  [299] = "0.269000,-22.048000,213.211000,-177.000000,0.007000,-179.714000,"
  [300] = "-1.345000,-22.065000,213.211000,-177.000000,-0.037000,178.570000,"
  [301] = "-2.959000,-22.137000,213.210000,-177.000000,-0.082000,176.853000,"
  [302] = "-4.573000,-22.261000,213.210000,-177.000000,-0.128000,175.133000,"
  [303] = "-6.186000,-22.440000,213.210000,-177.000000,-0.173000,173.409000,"
  [304] = "-7.799000,-22.673000,213.209000,-177.000000,-0.218000,171.678000,"
  [305] = "-9.410000,-22.962000,213.208000,-177.000000,-0.264000,169.940000,"
  [306] = "-11.020000,-23.306000,213.207000,-177.000000,-0.310000,168.192000,"
  [307] = "-12.628000,-23.707000,213.206000,-177.000000,-0.357000,166.434000,"
  [308] = "-14.234000,-24.166000,213.205000,-177.000000,-0.404000,164.662000,"
  [309] = "-15.838000,-24.685000,213.204000,-177.000000,-0.452000,162.874000,"
  [310] = "-17.439000,-25.265000,213.203000,-177.000000,-0.500000,161.070000,"
  [311] = "-17.459000,-25.264000,210.801000,-177.000000,-0.500000,161.072000,"
  [312] = "-17.480000,-25.264000,208.203000,-177.000000,-0.500000,161.074000,"
  [313] = "-16.142000,-24.776000,208.204000,-177.000000,-0.460000,162.579000,"
  [314] = "-14.535000,-24.248000,208.205000,-177.000000,-0.412000,164.368000,"
  [315] = "-12.925000,-23.779000,208.206000,-177.000000,-0.365000,166.142000,"
  [316] = "-11.313000,-23.368000,208.207000,-177.000000,-0.318000,167.903000,"
  [317] = "-9.700000,-23.015000,208.208000,-177.000000,-0.272000,169.652000,"
  [318] = "-8.085000,-22.717000,208.209000,-177.000000,-0.226000,171.391000,"
  [319] = "-6.470000,-22.475000,208.210000,-177.000000,-0.180000,173.122000,"
  [320] = "-4.853000,-22.287000,208.210000,-177.000000,-0.135000,174.847000,"
  [321] = "-3.236000,-22.154000,208.210000,-177.000000,-0.090000,176.567000,"
  [322] = "-1.618000,-22.074000,208.211000,-177.000000,-0.045000,178.284000,"
  [323] = "0.000000,-22.047000,208.211000,-177.000000,0.000000,180.000000,"
  [324] = "1.618000,-22.074000,208.211000,-177.000000,0.045000,-178.284000,"
  [325] = "3.236000,-22.154000,208.210000,-177.000000,0.090000,-176.567000,"
  [326] = "4.853000,-22.287000,208.210000,-177.000000,0.135000,-174.847000,"
  [327] = "6.470000,-22.475000,208.210000,-177.000000,0.180000,-173.122000,"
  [328] = "8.085000,-22.717000,208.209000,-177.000000,0.226000,-171.391000,"
  [329] = "9.700000,-23.015000,208.208000,-177.000000,0.272000,-169.651000,"
  [330] = "11.313000,-23.368000,208.207000,-177.000000,0.318000,-167.902000,"
  [331] = "12.925000,-23.779000,208.206000,-177.000000,0.365000,-166.142000,"
  [332] = "14.535000,-24.248000,208.205000,-177.000000,0.412000,-164.368000,"
  [333] = "16.142000,-24.776000,208.204000,-177.000000,0.460000,-162.579000,"
  [334] = "17.480000,-25.264000,208.203000,-177.000000,0.500000,-161.074000,"
  [335] = "17.502000,-25.264000,205.801000,-177.000000,0.500000,-161.072000,"
  [336] = "17.527000,-25.265000,203.203000,-177.000000,0.500000,-161.070000,"
  [337] = "15.929000,-24.689000,203.204000,-177.000000,0.452000,-162.861000,"
  [338] = "14.329000,-24.174000,203.206000,-177.000000,0.405000,-164.635000,"
  [339] = "12.727000,-23.717000,203.207000,-177.000000,0.358000,-166.393000,"
  [340] = "11.123000,-23.317000,203.208000,-177.000000,0.312000,-168.139000,"
  [341] = "9.518000,-22.974000,203.208000,-177.000000,0.266000,-169.874000,"
  [342] = "7.911000,-22.685000,203.209000,-177.000000,0.220000,-171.599000,"
  [343] = "6.303000,-22.451000,203.210000,-177.000000,0.175000,-173.316000,"
  [344] = "4.695000,-22.271000,203.210000,-177.000000,0.130000,-175.028000,"
  [345] = "3.085000,-22.144000,203.210000,-177.000000,0.086000,-176.735000,"
  [346] = "1.476000,-22.069000,203.211000,-177.000000,0.041000,-178.439000,"
  [347] = "0.134000,-22.047000,203.211000,-177.000000,0.004000,-179.858000,"
  [348] = "-1.476000,-22.069000,203.211000,-177.000000,-0.041000,178.439000,"
  [349] = "-3.085000,-22.144000,203.210000,-177.000000,-0.086000,176.735000,"
  [350] = "-4.695000,-22.271000,203.210000,-177.000000,-0.130000,175.028000,"
  [351] = "-6.303000,-22.451000,203.210000,-177.000000,-0.175000,173.316000,"
  [352] = "-7.911000,-22.685000,203.209000,-177.000000,-0.220000,171.599000,"
  [353] = "-9.518000,-22.974000,203.208000,-177.000000,-0.266000,169.874000,"
  [354] = "-11.123000,-23.317000,203.208000,-177.000000,-0.312000,168.139000,"
  [355] = "-12.727000,-23.717000,203.207000,-177.000000,-0.358000,166.393000,"
  [356] = "-14.329000,-24.174000,203.206000,-177.000000,-0.405000,164.635000,"
  [357] = "-15.929000,-24.689000,203.204000,-177.000000,-0.452000,162.861000,"
  [358] = "-17.527000,-25.265000,203.203000,-177.000000,-0.500000,161.070000,"
  [359] = "-17.546000,-25.264000,200.801000,-177.000000,-0.500000,161.072000,"
  [360] = "-17.567000,-25.264000,198.203000,-177.000000,-0.500000,161.074000,"
  [361] = "-15.966000,-24.688000,198.204000,-177.000000,-0.452000,162.864000,"
  [362] = "-14.362000,-24.173000,198.206000,-177.000000,-0.405000,164.638000,"
  [363] = "-12.756000,-23.716000,198.207000,-177.000000,-0.358000,166.396000,"
  [364] = "-11.148000,-23.317000,198.208000,-177.000000,-0.312000,168.141000,"
  [365] = "-9.539000,-22.973000,198.208000,-177.000000,-0.266000,169.876000,"
  [366] = "-7.929000,-22.685000,198.209000,-177.000000,-0.220000,171.600000,"
  [367] = "-6.317000,-22.451000,198.210000,-177.000000,-0.175000,173.318000,"
  [368] = "-4.705000,-22.271000,198.210000,-177.000000,-0.130000,175.029000,"
  [369] = "-3.092000,-22.143000,198.210000,-177.000000,-0.086000,176.736000,"
  [370] = "-1.479000,-22.069000,198.211000,-177.000000,-0.041000,178.439000,"
  [371] = "-0.134000,-22.047000,198.211000,-177.000000,-0.004000,179.858000,"
  [372] = "1.479000,-22.069000,198.211000,-177.000000,0.041000,-178.439000,"
  [373] = "3.092000,-22.143000,198.210000,-177.000000,0.086000,-176.736000,"
  [374] = "4.705000,-22.271000,198.210000,-177.000000,0.130000,-175.029000,"
  [375] = "6.317000,-22.451000,198.210000,-177.000000,0.175000,-173.318000,"
  [376] = "7.929000,-22.685000,198.209000,-177.000000,0.220000,-171.600000,"
  [377] = "9.539000,-22.973000,198.208000,-177.000000,0.266000,-169.875000,"
  [378] = "11.148000,-23.317000,198.208000,-177.000000,0.312000,-168.141000,"
  [379] = "12.756000,-23.716000,198.207000,-177.000000,0.358000,-166.396000,"
  [380] = "14.362000,-24.173000,198.206000,-177.000000,0.405000,-164.638000,"
  [381] = "15.966000,-24.688000,198.204000,-177.000000,0.452000,-162.864000,"
  [382] = "17.567000,-25.264000,198.203000,-177.000000,0.500000,-161.074000,"
  [383] = "17.590000,-25.264000,195.801000,-177.000000,0.500000,-161.072000,"
  [384] = "17.614000,-25.265000,193.203000,-177.000000,0.500000,-161.070000,"
  [385] = "16.008000,-24.689000,193.205000,-177.000000,0.452000,-162.861000,"
  [386] = "14.400000,-24.174000,193.206000,-177.000000,0.405000,-164.635000,"
  [387] = "12.790000,-23.717000,193.207000,-177.000000,0.358000,-166.393000,"
  [388] = "11.178000,-23.317000,193.208000,-177.000000,0.312000,-168.139000,"
  [389] = "9.564000,-22.974000,193.209000,-177.000000,0.266000,-169.874000,"
  [390] = "7.949000,-22.685000,193.209000,-177.000000,0.220000,-171.599000,"
  [391] = "6.334000,-22.451000,193.210000,-177.000000,0.175000,-173.316000,"
  [392] = "4.717000,-22.271000,193.210000,-177.000000,0.130000,-175.028000,"
  [393] = "3.100000,-22.143000,193.210000,-177.000000,0.086000,-176.735000,"
  [394] = "1.483000,-22.069000,193.211000,-177.000000,0.041000,-178.439000,"
  [395] = "0.135000,-22.047000,193.211000,-177.000000,0.004000,-179.858000,"
  [396] = "-1.483000,-22.069000,193.211000,-177.000000,-0.041000,178.439000,"
  [397] = "-3.100000,-22.144000,193.210000,-177.000000,-0.086000,176.735000,"
  [398] = "-4.717000,-22.271000,193.210000,-177.000000,-0.130000,175.028000,"
  [399] = "-6.334000,-22.451000,193.210000,-177.000000,-0.175000,173.316000,"
  [400] = "-7.949000,-22.685000,193.209000,-177.000000,-0.220000,171.599000,"
  [401] = "-9.564000,-22.974000,193.209000,-177.000000,-0.266000,169.874000,"
  [402] = "-11.178000,-23.317000,193.208000,-177.000000,-0.312000,168.139000,"
  [403] = "-12.790000,-23.717000,193.207000,-177.000000,-0.358000,166.393000,"
  [404] = "-14.400000,-24.174000,193.206000,-177.000000,-0.405000,164.635000,"
  [405] = "-16.008000,-24.689000,193.205000,-177.000000,-0.452000,162.861000,"
  [406] = "-17.614000,-25.265000,193.203000,-177.000000,-0.500000,161.070000,"
  [407] = "-17.633000,-25.264000,190.801000,-177.000000,-0.500000,161.072000,"
  [408] = "-17.654000,-25.264000,188.204000,-177.000000,-0.500000,161.074000,"
  [409] = "-16.057000,-24.692000,188.205000,-177.000000,-0.452000,162.851000,"
  [410] = "-14.457000,-24.180000,188.206000,-177.000000,-0.405000,164.611000,"
  [411] = "-12.855000,-23.726000,188.207000,-177.000000,-0.359000,166.356000,"
  [412] = "-11.252000,-23.328000,188.208000,-177.000000,-0.313000,168.089000,"
  [413] = "-9.647000,-22.985000,188.209000,-177.000000,-0.268000,169.810000,"
  [414] = "-8.041000,-22.697000,188.209000,-177.000000,-0.222000,171.522000,"
  [415] = "-6.434000,-22.462000,188.210000,-177.000000,-0.178000,173.227000,"
  [416] = "-4.826000,-22.280000,188.210000,-177.000000,-0.133000,174.925000,"
  [417] = "-3.218000,-22.150000,188.210000,-177.000000,-0.089000,176.619000,"
  [418] = "-1.609000,-22.073000,188.211000,-177.000000,-0.044000,178.310000,"
  [419] = "0.000000,-22.047000,188.211000,-177.000000,0.000000,180.000000,"
  [420] = "1.609000,-22.073000,188.211000,-177.000000,0.044000,-178.310000,"
  [421] = "3.218000,-22.150000,188.210000,-177.000000,0.089000,-176.619000,"
  [422] = "4.826000,-22.280000,188.210000,-177.000000,0.133000,-174.925000,"
  [423] = "6.434000,-22.462000,188.210000,-177.000000,0.178000,-173.227000,"
  [424] = "8.041000,-22.697000,188.209000,-177.000000,0.222000,-171.522000,"
  [425] = "9.647000,-22.985000,188.209000,-177.000000,0.268000,-169.810000,"
  [426] = "11.252000,-23.328000,188.208000,-177.000000,0.313000,-168.089000,"
  [427] = "12.855000,-23.726000,188.207000,-177.000000,0.359000,-166.356000,"
  [428] = "14.457000,-24.180000,188.206000,-177.000000,0.405000,-164.611000,"
  [429] = "16.057000,-24.692000,188.205000,-177.000000,0.452000,-162.851000,"
  [430] = "17.654000,-25.264000,188.204000,-177.000000,0.500000,-161.074000,"
  [431] = "17.677000,-25.264000,185.801000,-177.000000,0.500000,-161.072000,"
  [432] = "17.702000,-25.265000,183.204000,-177.000000,0.500000,-161.070000,"
  [433] = "16.099000,-24.693000,183.205000,-177.000000,0.453000,-162.847000,"
  [434] = "14.495000,-24.181000,183.206000,-177.000000,0.406000,-164.608000,"
  [435] = "12.889000,-23.727000,183.207000,-177.000000,0.359000,-166.354000,"
  [436] = "11.281000,-23.329000,183.208000,-177.000000,0.313000,-168.086000,"
  [437] = "9.672000,-22.986000,183.209000,-177.000000,0.268000,-169.808000,"
  [438] = "8.062000,-22.697000,183.209000,-177.000000,0.222000,-171.521000,"
  [439] = "6.450000,-22.462000,183.210000,-177.000000,0.178000,-173.225000,"
  [440] = "4.839000,-22.280000,183.210000,-177.000000,0.133000,-174.924000,"
  [441] = "3.226000,-22.151000,183.210000,-177.000000,0.089000,-176.619000,"
  [442] = "1.613000,-22.073000,183.211000,-177.000000,0.044000,-178.310000,"
  [443] = "0.000000,-22.047000,183.211000,-177.000000,0.000000,180.000000,"
  [444] = "-1.613000,-22.073000,183.211000,-177.000000,-0.044000,178.310000,"
  [445] = "-3.226000,-22.151000,183.210000,-177.000000,-0.089000,176.619000,"
  [446] = "-4.838000,-22.280000,183.210000,-177.000000,-0.133000,174.924000,"
  [447] = "-6.450000,-22.462000,183.210000,-177.000000,-0.178000,173.225000,"
  [448] = "-8.062000,-22.697000,183.209000,-177.000000,-0.222000,171.521000,"
  [449] = "-9.672000,-22.986000,183.209000,-177.000000,-0.268000,169.808000,"
  [450] = "-11.281000,-23.329000,183.208000,-177.000000,-0.313000,168.086000,"
  [451] = "-12.889000,-23.727000,183.207000,-177.000000,-0.359000,166.354000,"
  [452] = "-14.495000,-24.181000,183.206000,-177.000000,-0.406000,164.608000,"
  [453] = "-16.099000,-24.693000,183.205000,-177.000000,-0.453000,162.847000,"
  [454] = "-17.701000,-25.265000,183.204000,-177.000000,-0.500000,161.070000,"
  [455] = "-17.721000,-25.264000,180.802000,-177.000000,-0.500000,161.072000,"
  [456] = "-17.742000,-25.264000,178.204000,-177.000000,-0.500000,161.074000,"
  [457] = "-16.136000,-24.692000,178.205000,-177.000000,-0.452000,162.851000,"
  [458] = "-14.528000,-24.180000,178.206000,-177.000000,-0.405000,164.611000,"
  [459] = "-12.918000,-23.726000,178.207000,-177.000000,-0.359000,166.356000,"
  [460] = "-11.306000,-23.328000,178.208000,-177.000000,-0.313000,168.089000,"
  [461] = "-9.693000,-22.985000,178.209000,-177.000000,-0.268000,169.810000,"
  [462] = "-8.080000,-22.697000,178.209000,-177.000000,-0.222000,171.522000,"
  [463] = "-6.465000,-22.462000,178.210000,-177.000000,-0.178000,173.227000,"
  [464] = "-4.849000,-22.280000,178.210000,-177.000000,-0.133000,174.925000,"
  [465] = "-3.233000,-22.150000,178.210000,-177.000000,-0.089000,176.619000,"
  [466] = "-1.617000,-22.073000,178.211000,-177.000000,-0.044000,178.310000,"
  [467] = "0.000000,-22.047000,178.211000,-177.000000,0.000000,180.000000,"
  [468] = "1.617000,-22.073000,178.211000,-177.000000,0.044000,-178.310000,"
  [469] = "3.233000,-22.150000,178.210000,-177.000000,0.089000,-176.619000,"
  [470] = "4.849000,-22.280000,178.210000,-177.000000,0.133000,-174.925000,"
  [471] = "6.465000,-22.462000,178.210000,-177.000000,0.178000,-173.227000,"
  [472] = "8.080000,-22.697000,178.209000,-177.000000,0.222000,-171.522000,"
  [473] = "9.694000,-22.985000,178.209000,-177.000000,0.268000,-169.810000,"
  [474] = "11.306000,-23.328000,178.208000,-177.000000,0.313000,-168.089000,"
  [475] = "12.918000,-23.726000,178.207000,-177.000000,0.359000,-166.356000,"
  [476] = "14.528000,-24.180000,178.206000,-177.000000,0.405000,-164.611000,"
  [477] = "16.136000,-24.692000,178.205000,-177.000000,0.452000,-162.851000,"
  [478] = "17.742000,-25.264000,178.204000,-177.000000,0.500000,-161.074000,"
  [479] = "17.764000,-25.264000,175.802000,-177.000000,0.500000,-161.072000,"
  [480] = "17.789000,-25.265000,173.204000,-177.000000,0.500000,-161.070000,"
  [481] = "16.178000,-24.693000,173.205000,-177.000000,0.453000,-162.848000,"
  [482] = "14.566000,-24.181000,173.206000,-177.000000,0.406000,-164.608000,"
  [483] = "12.952000,-23.727000,173.207000,-177.000000,0.359000,-166.354000,"
  [484] = "11.336000,-23.329000,173.208000,-177.000000,0.313000,-168.086000,"
  [485] = "9.719000,-22.986000,173.209000,-177.000000,0.268000,-169.808000,"
  [486] = "8.101000,-22.697000,173.209000,-177.000000,0.222000,-171.521000,"
  [487] = "6.481000,-22.462000,173.210000,-177.000000,0.178000,-173.225000,"
  [488] = "4.862000,-22.280000,173.210000,-177.000000,0.133000,-174.924000,"
  [489] = "3.241000,-22.150000,173.210000,-177.000000,0.089000,-176.619000,"
  [490] = "1.621000,-22.073000,173.211000,-177.000000,0.044000,-178.310000,"
  [491] = "0.000000,-22.047000,173.211000,-177.000000,0.000000,180.000000,"
  [492] = "-1.621000,-22.073000,173.211000,-177.000000,-0.044000,178.310000,"
  [493] = "-3.241000,-22.151000,173.210000,-177.000000,-0.089000,176.619000,"
  [494] = "-4.862000,-22.280000,173.210000,-177.000000,-0.133000,174.924000,"
  [495] = "-6.481000,-22.462000,173.210000,-177.000000,-0.178000,173.225000,"
  [496] = "-8.101000,-22.697000,173.209000,-177.000000,-0.222000,171.521000,"
  [497] = "-9.719000,-22.986000,173.209000,-177.000000,-0.268000,169.808000,"
  [498] = "-11.336000,-23.329000,173.208000,-177.000000,-0.313000,168.086000,"
  [499] = "-12.952000,-23.727000,173.207000,-177.000000,-0.359000,166.354000,"
  [500] = "-14.566000,-24.181000,173.206000,-177.000000,-0.406000,164.608000,"
  [501] = "-16.178000,-24.693000,173.205000,-177.000000,-0.453000,162.848000,"
  [502] = "-17.789000,-25.265000,173.204000,-177.000000,-0.500000,161.070000,"
  [503] = "-17.808000,-25.264000,170.802000,-177.000000,-0.500000,161.072000,"
  [504] = "-17.829000,-25.264000,168.204000,-177.000000,-0.500000,161.074000,"
  [505] = "-16.227000,-24.696000,168.205000,-177.000000,-0.453000,162.838000,"
  [506] = "-14.623000,-24.188000,168.206000,-177.000000,-0.406000,164.585000,"
  [507] = "-13.017000,-23.736000,168.207000,-177.000000,-0.360000,166.317000,"
  [508] = "-11.410000,-23.339000,168.208000,-177.000000,-0.314000,168.037000,"
  [509] = "-9.801000,-22.997000,168.209000,-177.000000,-0.269000,169.746000,"
  [510] = "-8.192000,-22.709000,168.209000,-177.000000,-0.224000,171.445000,"
  [511] = "-6.581000,-22.473000,168.210000,-177.000000,-0.180000,173.137000,"
  [512] = "-4.970000,-22.290000,168.210000,-177.000000,-0.136000,174.823000,"
  [513] = "-3.358000,-22.158000,168.210000,-177.000000,-0.092000,176.505000,"
  [514] = "-1.746000,-22.077000,168.211000,-177.000000,-0.048000,178.183000,"
  [515] = "-0.672000,-22.051000,168.211000,-177.000000,-0.018000,179.301000,"
  [516] = "0.134000,-22.047000,168.211000,-177.000000,0.004000,-179.860000,"
  [517] = "1.747000,-22.077000,168.211000,-177.000000,0.048000,-178.183000,"
  [518] = "3.358000,-22.158000,168.210000,-177.000000,0.092000,-176.505000,"
  [519] = "4.970000,-22.290000,168.210000,-177.000000,0.136000,-174.823000,"
  [520] = "6.581000,-22.473000,168.210000,-177.000000,0.180000,-173.137000,"
  [521] = "8.192000,-22.709000,168.209000,-177.000000,0.224000,-171.445000,"
  [522] = "9.801000,-22.997000,168.209000,-177.000000,0.269000,-169.746000,"
  [523] = "11.410000,-23.339000,168.208000,-177.000000,0.314000,-168.037000,"
  [524] = "13.017000,-23.736000,168.207000,-177.000000,0.360000,-166.317000,"
  [525] = "14.623000,-24.188000,168.206000,-177.000000,0.406000,-164.585000,"
  [526] = "16.227000,-24.696000,168.205000,-177.000000,0.453000,-162.838000,"
  [527] = "17.829000,-25.264000,168.204000,-177.000000,0.500000,-161.074000,"
  [528] = "17.852000,-25.264000,165.802000,-177.000000,0.500000,-161.072000,"
  [529] = "17.876000,-25.265000,163.204000,-177.000000,0.500000,-161.070000,"
  [530] = "16.270000,-24.697000,163.206000,-177.000000,0.453000,-162.834000,"
  [531] = "14.661000,-24.188000,163.207000,-177.000000,0.406000,-164.582000,"
  [532] = "13.051000,-23.736000,163.207000,-177.000000,0.360000,-166.314000,"
  [533] = "11.439000,-23.340000,163.208000,-177.000000,0.314000,-168.034000,"
  [534] = "9.827000,-22.998000,163.209000,-177.000000,0.269000,-169.744000,"
  [535] = "8.213000,-22.709000,163.209000,-177.000000,0.224000,-171.444000,"
  [536] = "6.598000,-22.473000,163.210000,-177.000000,0.180000,-173.136000,"
  [537] = "4.983000,-22.290000,163.210000,-177.000000,0.136000,-174.822000,"
  [538] = "3.367000,-22.158000,163.210000,-177.000000,0.092000,-176.504000,"
  [539] = "1.751000,-22.077000,163.211000,-177.000000,0.048000,-178.183000,"
  [540] = "0.673000,-22.051000,163.211000,-177.000000,0.018000,-179.301000,"
  [541] = "-0.135000,-22.047000,163.211000,-177.000000,-0.004000,179.860000,"
  [542] = "-1.751000,-22.077000,163.211000,-177.000000,-0.048000,178.183000,"
  [543] = "-3.367000,-22.158000,163.210000,-177.000000,-0.092000,176.504000,"
  [544] = "-4.983000,-22.290000,163.210000,-177.000000,-0.136000,174.822000,"
  [545] = "-6.598000,-22.473000,163.210000,-177.000000,-0.180000,173.136000,"
  [546] = "-8.213000,-22.709000,163.209000,-177.000000,-0.224000,171.444000,"
  [547] = "-9.827000,-22.998000,163.209000,-177.000000,-0.269000,169.744000,"
  [548] = "-11.439000,-23.340000,163.208000,-177.000000,-0.314000,168.034000,"
  [549] = "-13.051000,-23.736000,163.207000,-177.000000,-0.360000,166.314000,"
  [550] = "-14.661000,-24.188000,163.207000,-177.000000,-0.406000,164.582000,"
  [551] = "-16.270000,-24.697000,163.206000,-177.000000,-0.453000,162.834000,"
  [552] = "-17.876000,-25.265000,163.204000,-177.000000,-0.500000,161.070000,"
  [553] = "-17.896000,-25.264000,160.802000,-177.000000,-0.500000,161.072000,"
  [554] = "-17.917000,-25.264000,158.205000,-177.000000,-0.500000,161.074000,"
  [555] = "-16.306000,-24.696000,158.206000,-177.000000,-0.453000,162.838000,"
  [556] = "-14.694000,-24.188000,158.207000,-177.000000,-0.406000,164.585000,"
  [557] = "-13.080000,-23.736000,158.208000,-177.000000,-0.360000,166.317000,"
  [558] = "-11.465000,-23.339000,158.208000,-177.000000,-0.314000,168.037000,"
  [559] = "-9.848000,-22.997000,158.209000,-177.000000,-0.269000,169.746000,"
  [560] = "-8.231000,-22.709000,158.209000,-177.000000,-0.224000,171.445000,"
  [561] = "-6.613000,-22.473000,158.210000,-177.000000,-0.180000,173.137000,"
  [562] = "-4.994000,-22.290000,158.210000,-177.000000,-0.136000,174.823000,"
  [563] = "-3.374000,-22.158000,158.210000,-177.000000,-0.092000,176.505000,"
  [564] = "-1.755000,-22.077000,158.211000,-177.000000,-0.048000,178.183000,"
  [565] = "-0.675000,-22.051000,158.211000,-177.000000,-0.018000,179.301000,"
  [566] = "0.135000,-22.047000,158.211000,-177.000000,0.004000,-179.860000,"
  [567] = "1.755000,-22.077000,158.211000,-177.000000,0.048000,-178.183000,"
  [568] = "3.374000,-22.158000,158.210000,-177.000000,0.092000,-176.505000,"
  [569] = "4.994000,-22.290000,158.210000,-177.000000,0.136000,-174.823000,"
  [570] = "6.613000,-22.473000,158.210000,-177.000000,0.180000,-173.137000,"
  [571] = "8.231000,-22.709000,158.209000,-177.000000,0.224000,-171.445000,"
  [572] = "9.848000,-22.997000,158.209000,-177.000000,0.269000,-169.746000,"
  [573] = "11.465000,-23.339000,158.208000,-177.000000,0.314000,-168.037000,"
  [574] = "13.080000,-23.736000,158.208000,-177.000000,0.360000,-166.317000,"
  [575] = "14.694000,-24.188000,158.207000,-177.000000,0.406000,-164.585000,"
  [576] = "16.306000,-24.696000,158.206000,-177.000000,0.453000,-162.838000,"
  [577] = "17.917000,-25.264000,158.205000,-177.000000,0.500000,-161.074000,"
  [578] = "17.939000,-25.264000,155.803000,-177.000000,0.500000,-161.072000,"
  [579] = "17.964000,-25.265000,153.205000,-177.000000,0.500000,-161.070000,"
  [580] = "16.361000,-24.701000,153.206000,-177.000000,0.453000,-162.821000,"
  [581] = "14.756000,-24.196000,153.207000,-177.000000,0.407000,-164.556000,"
  [582] = "13.150000,-23.746000,153.208000,-177.000000,0.361000,-166.276000,"
  [583] = "11.543000,-23.351000,153.208000,-177.000000,0.316000,-167.983000,"
  [584] = "9.934000,-23.010000,153.209000,-177.000000,0.271000,-169.680000,"
  [585] = "8.325000,-22.721000,153.209000,-177.000000,0.226000,-171.368000,"
  [586] = "6.714000,-22.484000,153.210000,-177.000000,0.182000,-173.048000,"
  [587] = "5.103000,-22.299000,153.210000,-177.000000,0.138000,-174.722000,"
  [588] = "3.492000,-22.165000,153.210000,-177.000000,0.095000,-176.391000,"
  [589] = "1.880000,-22.081000,153.211000,-177.000000,0.051000,-178.058000,"
  [590] = "0.806000,-22.053000,153.211000,-177.000000,0.022000,-179.168000,"
  [591] = "-0.269000,-22.048000,153.211000,-177.000000,-0.007000,179.723000,"
  [592] = "-1.880000,-22.081000,153.211000,-177.000000,-0.051000,178.058000,"
  [593] = "-3.492000,-22.165000,153.210000,-177.000000,-0.095000,176.391000,"
  [594] = "-5.103000,-22.299000,153.210000,-177.000000,-0.138000,174.722000,"
  [595] = "-6.714000,-22.484000,153.210000,-177.000000,-0.182000,173.048000,"
  [596] = "-8.325000,-22.721000,153.209000,-177.000000,-0.226000,171.368000,"
  [597] = "-9.934000,-23.010000,153.209000,-177.000000,-0.271000,169.680000,"
  [598] = "-11.543000,-23.351000,153.208000,-177.000000,-0.316000,167.983000,"
  [599] = "-13.150000,-23.746000,153.208000,-177.000000,-0.361000,166.276000,"
  [600] = "-14.756000,-24.196000,153.207000,-177.000000,-0.407000,164.556000,"
  [601] = "-16.361000,-24.701000,153.206000,-177.000000,-0.453000,162.821000,"
  [602] = "-17.964000,-25.265000,153.205000,-177.000000,-0.500000,161.070000,"
  [603] = "-17.983000,-25.264000,150.803000,-177.000000,-0.500000,161.072000,"
  [604] = "-18.004000,-25.264000,148.205000,-177.000000,-0.500000,161.074000,"
  [605] = "-16.397000,-24.700000,148.206000,-177.000000,-0.453000,162.825000,"
  [606] = "-14.789000,-24.195000,148.207000,-177.000000,-0.407000,164.559000,"
  [607] = "-13.179000,-23.745000,148.208000,-177.000000,-0.361000,166.279000,"
  [608] = "-11.568000,-23.350000,148.208000,-177.000000,-0.316000,167.986000,"
  [609] = "-9.956000,-23.009000,148.209000,-177.000000,-0.271000,169.682000,"
  [610] = "-8.343000,-22.721000,148.209000,-177.000000,-0.226000,171.369000,"
  [611] = "-6.729000,-22.484000,148.210000,-177.000000,-0.182000,173.049000,"
  [612] = "-5.115000,-22.299000,148.210000,-177.000000,-0.138000,174.723000,"
  [613] = "-3.500000,-22.165000,148.210000,-177.000000,-0.095000,176.392000,"
  [614] = "-1.885000,-22.081000,148.211000,-177.000000,-0.051000,178.058000,"
  [615] = "-0.808000,-22.053000,148.211000,-177.000000,-0.022000,179.168000,"
  [616] = "0.269000,-22.048000,148.211000,-177.000000,0.007000,-179.723000,"
  [617] = "1.885000,-22.081000,148.211000,-177.000000,0.051000,-178.058000,"
  [618] = "3.500000,-22.165000,148.210000,-177.000000,0.095000,-176.392000,"
  [619] = "5.115000,-22.299000,148.210000,-177.000000,0.138000,-174.723000,"
  [620] = "6.729000,-22.484000,148.210000,-177.000000,0.182000,-173.049000,"
  [621] = "8.343000,-22.721000,148.209000,-177.000000,0.226000,-171.369000,"
  [622] = "9.956000,-23.009000,148.209000,-177.000000,0.271000,-169.682000,"
  [623] = "11.568000,-23.350000,148.208000,-177.000000,0.316000,-167.986000,"
  [624] = "13.179000,-23.745000,148.208000,-177.000000,0.361000,-166.278000,"
  [625] = "14.789000,-24.195000,148.207000,-177.000000,0.407000,-164.559000,"
  [626] = "16.397000,-24.700000,148.206000,-177.000000,0.453000,-162.825000,"
  [627] = "18.004000,-25.264000,148.205000,-177.000000,0.500000,-161.074000,"
  [628] = "18.027000,-25.264000,145.803000,-177.000000,0.500000,-161.072000,"
  [629] = "18.051000,-25.265000,143.205000,-177.000000,0.500000,-161.070000,"
  [630] = "16.440000,-24.701000,143.206000,-177.000000,0.453000,-162.821000,"
  [631] = "14.827000,-24.196000,143.207000,-177.000000,0.407000,-164.556000,"
  [632] = "13.213000,-23.746000,143.208000,-177.000000,0.361000,-166.276000,"
  [633] = "11.598000,-23.351000,143.208000,-177.000000,0.316000,-167.983000,"
  [634] = "9.981000,-23.009000,143.209000,-177.000000,0.271000,-169.680000,"
  [635] = "8.364000,-22.721000,143.209000,-177.000000,0.226000,-171.368000,"
  [636] = "6.746000,-22.484000,143.210000,-177.000000,0.182000,-173.048000,"
  [637] = "5.128000,-22.299000,143.210000,-177.000000,0.138000,-174.722000,"
  [638] = "3.509000,-22.165000,143.210000,-177.000000,0.095000,-176.391000,"
  [639] = "1.889000,-22.081000,143.211000,-177.000000,0.051000,-178.058000,"
  [640] = "0.810000,-22.053000,143.211000,-177.000000,0.022000,-179.168000,"
  [641] = "-0.270000,-22.048000,143.211000,-177.000000,-0.007000,179.723000,"
  [642] = "-1.889000,-22.081000,143.211000,-177.000000,-0.051000,178.058000,"
  [643] = "-3.509000,-22.165000,143.210000,-177.000000,-0.095000,176.391000,"
  [644] = "-5.128000,-22.299000,143.210000,-177.000000,-0.138000,174.722000,"
  [645] = "-6.746000,-22.484000,143.210000,-177.000000,-0.182000,173.048000,"
  [646] = "-8.364000,-22.721000,143.209000,-177.000000,-0.226000,171.368000,"
  [647] = "-9.981000,-23.010000,143.209000,-177.000000,-0.271000,169.680000,"
  [648] = "-11.598000,-23.351000,143.208000,-177.000000,-0.316000,167.983000,"
  [649] = "-13.213000,-23.746000,143.208000,-177.000000,-0.361000,166.276000,"
  [650] = "-14.827000,-24.196000,143.207000,-177.000000,-0.407000,164.556000,"
  [651] = "-16.440000,-24.701000,143.206000,-177.000000,-0.453000,162.821000,"
  [652] = "-18.051000,-25.265000,143.205000,-177.000000,-0.500000,161.071000,"
  [653] = "-18.070000,-25.264000,140.803000,-177.000000,-0.500000,161.072000,"
  [654] = "-18.091000,-25.264000,138.205000,-177.000000,-0.500000,161.074000,"
  [655] = "-16.537000,-24.720000,138.206000,-177.000000,-0.455000,162.760000,"
  [656] = "-15.025000,-24.244000,138.207000,-177.000000,-0.412000,164.383000,"
  [657] = "-13.512000,-23.816000,138.208000,-177.000000,-0.369000,165.993000,"
  [658] = "-11.860000,-23.405000,138.208000,-177.000000,-0.322000,167.737000,"
  [659] = "-10.207000,-23.049000,138.209000,-177.000000,-0.277000,169.469000,"
  [660] = "-8.553000,-22.749000,138.209000,-177.000000,-0.231000,171.192000,"
  [661] = "-6.899000,-22.502000,138.210000,-177.000000,-0.186000,172.906000,"
  [662] = "-5.244000,-22.310000,138.210000,-177.000000,-0.141000,174.615000,"
  [663] = "-3.588000,-22.170000,138.210000,-177.000000,-0.096000,176.318000,"
  [664] = "-1.932000,-22.082000,138.211000,-177.000000,-0.052000,178.018000,"
  [665] = "-0.828000,-22.053000,138.211000,-177.000000,-0.022000,179.151000,"
  [666] = "0.276000,-22.048000,138.211000,-177.000000,0.007000,-179.717000,"
  [667] = "1.932000,-22.082000,138.211000,-177.000000,0.052000,-178.018000,"
  [668] = "3.588000,-22.170000,138.210000,-177.000000,0.096000,-176.318000,"
  [669] = "5.244000,-22.310000,138.210000,-177.000000,0.141000,-174.615000,"
  [670] = "6.899000,-22.502000,138.210000,-177.000000,0.186000,-172.906000,"
  [671] = "8.553000,-22.749000,138.209000,-177.000000,0.231000,-171.192000,"
  [672] = "10.207000,-23.049000,138.209000,-177.000000,0.277000,-169.469000,"
  [673] = "11.860000,-23.405000,138.208000,-177.000000,0.322000,-167.737000,"
  [674] = "13.512000,-23.816000,138.208000,-177.000000,0.369000,-165.993000,"
  [675] = "15.025000,-24.244000,138.207000,-177.000000,0.412000,-164.383000,"
  [676] = "16.537000,-24.720000,138.206000,-177.000000,0.455000,-162.759000,"
  [677] = "18.091000,-25.264000,138.205000,-177.000000,0.500000,-161.074000,"
  [678] = "18.114000,-25.264000,135.803000,-177.000000,0.500000,-161.072000,"
  [679] = "18.138000,-25.265000,133.206000,-177.000000,0.500000,-161.071000,"
  [680] = "16.531000,-24.705000,133.206000,-177.000000,0.454000,-162.809000,"
  [681] = "14.922000,-24.203000,133.207000,-177.000000,0.408000,-164.530000,"
  [682] = "13.312000,-23.755000,133.208000,-177.000000,0.362000,-166.238000,"
  [683] = "11.701000,-23.362000,133.209000,-177.000000,0.317000,-167.933000,"
  [684] = "10.089000,-23.021000,133.209000,-177.000000,0.273000,-169.617000,"
  [685] = "8.476000,-22.733000,133.210000,-177.000000,0.228000,-171.293000,"
  [686] = "6.862000,-22.495000,133.210000,-177.000000,0.185000,-172.961000,"
  [687] = "5.248000,-22.309000,133.210000,-177.000000,0.141000,-174.623000,"
  [688] = "3.634000,-22.172000,133.210000,-177.000000,0.097000,-176.280000,"
  [689] = "2.019000,-22.086000,133.211000,-177.000000,0.054000,-177.934000,"
  [690] = "0.673000,-22.051000,133.211000,-177.000000,0.018000,-179.312000,"
  [691] = "-0.404000,-22.048000,133.211000,-177.000000,-0.011000,179.587000,"
  [692] = "-2.019000,-22.086000,133.211000,-177.000000,-0.054000,177.934000,"
  [693] = "-3.634000,-22.172000,133.210000,-177.000000,-0.097000,176.280000,"
  [694] = "-5.248000,-22.309000,133.210000,-177.000000,-0.141000,174.623000,"
  [695] = "-6.862000,-22.495000,133.210000,-177.000000,-0.185000,172.961000,"
  [696] = "-8.476000,-22.733000,133.210000,-177.000000,-0.228000,171.293000,"
  [697] = "-10.089000,-23.021000,133.209000,-177.000000,-0.273000,169.617000,"
  [698] = "-11.701000,-23.362000,133.209000,-177.000000,-0.317000,167.933000,"
  [699] = "-13.312000,-23.755000,133.208000,-177.000000,-0.362000,166.238000,"
  [700] = "-14.922000,-24.203000,133.207000,-177.000000,-0.408000,164.530000,"
  [701] = "-16.531000,-24.705000,133.206000,-177.000000,-0.454000,162.809000,"
  [702] = "-18.138000,-25.265000,133.206000,-177.000000,-0.500000,161.071000,"
  [703] = "-18.162000,-25.265000,130.659000,-177.000000,-0.500000,161.069000,"
  [704] = "-16.552000,-24.706000,130.660000,-177.000000,-0.454000,162.808000,"
  [705] = "-14.941000,-24.203000,130.661000,-177.000000,-0.408000,164.529000,"
  [706] = "-13.329000,-23.755000,130.662000,-177.000000,-0.362000,166.237000,"
  [707] = "-11.716000,-23.362000,130.662000,-177.000000,-0.317000,167.932000,"
  [708] = "-10.102000,-23.021000,130.663000,-177.000000,-0.273000,169.617000,"
  [709] = "-8.487000,-22.733000,130.663000,-177.000000,-0.228000,171.292000,"
  [710] = "-6.871000,-22.495000,130.663000,-177.000000,-0.185000,172.960000,"
  [711] = "-5.255000,-22.309000,130.664000,-177.000000,-0.141000,174.622000,"
  [712] = "-3.638000,-22.172000,130.664000,-177.000000,-0.097000,176.280000,"
  [713] = "-2.021000,-22.086000,130.664000,-177.000000,-0.054000,177.934000,"
  [714] = "-0.674000,-22.051000,130.664000,-177.000000,-0.018000,179.312000,"
  [715] = "0.404000,-22.048000,130.664000,-177.000000,0.011000,-179.587000,"
  [716] = "2.021000,-22.086000,130.664000,-177.000000,0.054000,-177.934000,"
  [717] = "3.638000,-22.172000,130.664000,-177.000000,0.097000,-176.280000,"
  [718] = "5.255000,-22.309000,130.664000,-177.000000,0.141000,-174.622000,"
  [719] = "6.871000,-22.495000,130.663000,-177.000000,0.185000,-172.960000,"
  [720] = "8.487000,-22.733000,130.663000,-177.000000,0.228000,-171.292000,"
  [721] = "10.102000,-23.021000,130.663000,-177.000000,0.273000,-169.617000,"
  [722] = "11.716000,-23.362000,130.662000,-177.000000,0.317000,-167.932000,"
  [723] = "13.329000,-23.755000,130.662000,-177.000000,0.362000,-166.237000,"
  [724] = "14.941000,-24.203000,130.661000,-177.000000,0.408000,-164.529000,"
  [725] = "16.552000,-24.706000,130.660000,-177.000000,0.454000,-162.807000,"
  [726] = "18.162000,-25.265000,130.659000,-177.000000,0.500000,-161.069000,"
  [727] = "18.185000,-25.266000,128.087000,-177.000000,0.500000,-161.069000,"
  [728] = "16.573000,-24.706000,128.088000,-177.000000,0.454000,-162.807000,"
  [729] = "14.960000,-24.203000,128.089000,-177.000000,0.408000,-164.529000,"
  [730] = "13.346000,-23.755000,128.090000,-177.000000,0.362000,-166.236000,"
  [731] = "11.731000,-23.362000,128.090000,-177.000000,0.317000,-167.932000,"
  [732] = "10.114000,-23.021000,128.091000,-177.000000,0.273000,-169.616000,"
  [733] = "8.497000,-22.733000,128.091000,-177.000000,0.228000,-171.292000,"
  [734] = "6.880000,-22.495000,128.092000,-177.000000,0.185000,-172.960000,"
  [735] = "5.261000,-22.309000,128.092000,-177.000000,0.141000,-174.622000,"
  [736] = "3.643000,-22.172000,128.092000,-177.000000,0.097000,-176.280000,"
  [737] = "2.024000,-22.086000,128.092000,-177.000000,0.054000,-177.934000,"
  [738] = "0.675000,-22.051000,128.092000,-177.000000,0.018000,-179.312000,"
  [739] = "-0.405000,-22.048000,128.092000,-177.000000,-0.011000,179.587000,"
  [740] = "-2.024000,-22.086000,128.092000,-177.000000,-0.054000,177.934000,"
  [741] = "-3.643000,-22.172000,128.092000,-177.000000,-0.097000,176.280000,"
  [742] = "-5.261000,-22.309000,128.092000,-177.000000,-0.141000,174.622000,"
  [743] = "-6.879000,-22.496000,128.092000,-177.000000,-0.185000,172.960000,"
  [744] = "-8.497000,-22.733000,128.091000,-177.000000,-0.228000,171.292000,"
  [745] = "-10.114000,-23.021000,128.091000,-177.000000,-0.273000,169.616000,"
  [746] = "-11.731000,-23.362000,128.090000,-177.000000,-0.317000,167.932000,"
  [747] = "-13.346000,-23.755000,128.090000,-177.000000,-0.362000,166.236000,"
  [748] = "-14.960000,-24.203000,128.089000,-177.000000,-0.408000,164.529000,"
  [749] = "-16.573000,-24.706000,128.088000,-177.000000,-0.454000,162.807000,"
  [750] = "-18.185000,-25.266000,128.087000,-177.000000,-0.500000,161.069000,"
  [751] = "-18.208000,-25.266000,125.490000,-177.000000,-0.500000,161.068000,"
  [752] = "-16.594000,-24.706000,125.491000,-177.000000,-0.454000,162.806000,"
  [753] = "-14.979000,-24.203000,125.491000,-177.000000,-0.408000,164.528000,"
  [754] = "-13.363000,-23.756000,125.492000,-177.000000,-0.362000,166.236000,"
  [755] = "-11.745000,-23.362000,125.493000,-177.000000,-0.317000,167.932000,"
  [756] = "-10.127000,-23.021000,125.493000,-177.000000,-0.273000,169.616000,"
  [757] = "-8.508000,-22.733000,125.494000,-177.000000,-0.228000,171.292000,"
  [758] = "-6.888000,-22.496000,125.494000,-177.000000,-0.185000,172.960000,"
  [759] = "-5.268000,-22.309000,125.494000,-177.000000,-0.141000,174.622000,"
  [760] = "-3.647000,-22.172000,125.494000,-177.000000,-0.097000,176.280000,"
  [761] = "-2.026000,-22.086000,125.495000,-177.000000,-0.054000,177.934000,"
  [762] = "-0.675000,-22.051000,125.495000,-177.000000,-0.018000,179.312000,"
  [763] = "0.405000,-22.048000,125.495000,-177.000000,0.011000,-179.587000,"
  [764] = "2.026000,-22.086000,125.495000,-177.000000,0.054000,-177.934000,"
  [765] = "3.647000,-22.172000,125.494000,-177.000000,0.097000,-176.280000,"
  [766] = "5.268000,-22.309000,125.494000,-177.000000,0.141000,-174.622000,"
  [767] = "6.888000,-22.496000,125.494000,-177.000000,0.185000,-172.960000,"
  [768] = "8.508000,-22.733000,125.494000,-177.000000,0.228000,-171.292000,"
  [769] = "10.127000,-23.021000,125.493000,-177.000000,0.273000,-169.616000,"
  [770] = "11.745000,-23.362000,125.493000,-177.000000,0.317000,-167.931000,"
  [771] = "13.363000,-23.756000,125.492000,-177.000000,0.362000,-166.236000,"
  [772] = "14.979000,-24.203000,125.491000,-177.000000,0.408000,-164.528000,"
  [773] = "16.594000,-24.706000,125.491000,-177.000000,0.454000,-162.806000,"
  [774] = "18.208000,-25.266000,125.490000,-177.000000,0.500000,-161.068000,"
  [775] = "18.225000,-25.264000,123.020000,-177.000000,0.500000,-161.073000,"
  [776] = "16.610000,-24.705000,123.021000,-177.000000,0.454000,-162.811000,"
  [777] = "14.993000,-24.202000,123.022000,-177.000000,0.408000,-164.532000,"
  [778] = "13.375000,-23.755000,123.022000,-177.000000,0.362000,-166.240000,"
  [779] = "11.756000,-23.361000,123.023000,-177.000000,0.317000,-167.935000,"
  [780] = "10.136000,-23.021000,123.023000,-177.000000,0.273000,-169.619000,"
  [781] = "8.515000,-22.732000,123.024000,-177.000000,0.228000,-171.294000,"
  [782] = "6.894000,-22.495000,123.024000,-177.000000,0.185000,-172.962000,"
  [783] = "5.273000,-22.309000,123.024000,-177.000000,0.141000,-174.623000,"
  [784] = "3.650000,-22.172000,123.025000,-177.000000,0.097000,-176.281000,"
  [785] = "2.028000,-22.086000,123.025000,-177.000000,0.054000,-177.935000,"
  [786] = "0.676000,-22.051000,123.025000,-177.000000,0.018000,-179.312000,"
  [787] = "-0.406000,-22.048000,123.025000,-177.000000,-0.011000,179.587000,"
  [788] = "-2.028000,-22.086000,123.025000,-177.000000,-0.054000,177.935000,"
  [789] = "-3.650000,-22.172000,123.025000,-177.000000,-0.097000,176.281000,"
  [790] = "-5.273000,-22.309000,123.024000,-177.000000,-0.141000,174.623000,"
  [791] = "-6.894000,-22.495000,123.024000,-177.000000,-0.185000,172.962000,"
  [792] = "-8.515000,-22.732000,123.024000,-177.000000,-0.228000,171.294000,"
  [793] = "-10.136000,-23.021000,123.023000,-177.000000,-0.273000,169.619000,"
  [794] = "-11.756000,-23.361000,123.023000,-177.000000,-0.317000,167.935000,"
  [795] = "-13.375000,-23.755000,123.022000,-177.000000,-0.362000,166.240000,"
  [796] = "-14.993000,-24.202000,123.022000,-177.000000,-0.408000,164.533000,"
  [797] = "-16.610000,-24.705000,123.021000,-177.000000,-0.454000,162.811000,"
  [798] = "-18.225000,-25.264000,123.020000,-177.000000,-0.500000,161.073000,"
tool tTool = {fatherId=flange[0], ioLink=valve1}
public sio sSocketout

--- initdata.pgx ---
program initdata()
begin
  nTxtTotal=11
  nNumTotal=5031
  n_sTxt=0
  nNumrecord=0
  fout=true
  bSignal=false
  bTxt1=false
  bTxt2=false
  bTxt3=false
  btrig=true
  call Txt_initData()
  call txt_PkgInit()

  //clearBuffer(sSocketout)
  //sioSet(sSocketout,nByteOut)
end

--- PositionTrigger.pgx ---
program PositionTrigger()
  local num nhere
begin
  ntime=clock()
  nnnn=0
  shere=pfrmCad[0]
  call Transmission()
  delay(0)
  while true
    if bSignal==true
      //shere=here(tTool,FrmDraw)
      shere=here(tTool,world)
      fout=false
      delay(0)
      fout=true
      delay(0.005)
      call Transmission()
      delay(0)
      ndelay=clock()-ntime
      nnnn=nnnn+1
    endIf
    delay(0)
  endWhile
  ndelay=clock()-ntime
end

--- Transmission.pgx ---
program Transmission()
  local num nByteOut[48]
  local num nTranC[6]
begin
  nTranC[0]=shere[0].trsf.x
  nTranC[1]=shere[0].trsf.y
  nTranC[2]=shere[0].trsf.z
  nTranC[3]=shere[0].trsf.rx
  nTranC[4]=shere[0].trsf.ry
  nTranC[5]=shere[0].trsf.rz
  toBinary(nTranC,6,"8.0b",nByteOut)
  sioSet(sSocketout,nByteOut)
end

--- Txt_initData.pgx ---
program Txt_initData()
begin
  while size(sString)>1
    $ddel(sString,size(sString)-1)
  endWhile
  while size(pfrmCad)>1
    $ddel(pfrmCad,size(pfrmCad)-1)
  endWhile
  sString[0]=""
  pfrmCad[0].trsf={0,0,0,0,0,0}
  for l_nInit=1 to 1499
    $dins(sString,l_nInit)
    $dins(pfrmCad,l_nInit)
  endFor
end

--- TxtReadRoom2.pgx ---
program TxtReadRoom2()
  local string l_str
  local num nNumpoint
  local num ntext
  local string sTxtfile
begin
  bTxt2=false
  delay(0)
  l_str=toString("1",n_sTxt)
  sTxtfile="path"+l_str+".txt"
  ntext=$fileOpen(sTxtfile,"r")
  for nNumpoint=500 to 999
    $fileGet(ntext,sString[nNumpoint],1)
    if sString[nNumpoint]!=""
      call stringtopoint(sString[nNumpoint],nNumpoint)
    else
    endIf
  endFor
  delay(0)

  if n_sTxt==nTxtTotal-1
    n_sTxt=0
  elseIf n_sTxt!=nTxtTotal-1
    n_sTxt=n_sTxt+1
  endIf
  nNumpoint=nNumpoint-1
  $fileClose(ntext)
end

--- TxtReadRoom3.pgx ---
program TxtReadRoom3()
  local string l_str
  local num nNumpoint
  local num ntext
  local string sTxtfile
begin
  bTxt3=false
  delay(0)
  l_str=toString("1",n_sTxt)
  sTxtfile="path"+l_str+".txt"
  ntext=$fileOpen(sTxtfile,"r")
  for nNumpoint=1000 to 1499
    $fileGet(ntext,sString[nNumpoint],1)
    if sString[nNumpoint]!=""
      call stringtopoint(sString[nNumpoint],nNumpoint)
    else
    endIf
  endFor
  delay(0)

  if n_sTxt==nTxtTotal-1
    n_sTxt=0
  elseIf n_sTxt!=nTxtTotal-1
    n_sTxt=n_sTxt+1
  endIf
  nNumpoint=nNumpoint-1
  $fileClose(ntext)
end

--- WipeCacheRoom1.pgx ---
program WipeCacheRoom1()
  local num nNum
begin

  for nNum=0 to 499
    sString[nNum]=""
    pfrmCad[nNum].trsf={0,0,0,0,0,0}
  endFor

end

--- WipeCacheRoom2.pgx ---
program WipeCacheRoom2()
  local num nNum
begin
  for nNum=500 to 999
    sString[nNum]=""
    pfrmCad[nNum].trsf={0,0,0,0,0,0}
  endFor

end
